FUNCTION_BLOCK FB_SLIDERLR (* FB_SLIDER with local publication of REAL position *)
  (* Standard: 61499-1; Classification: HMI *)
  (* Version 0.0, 2006-11-15, JHC, Holobloc Inc, Copied/Modified from FB_SLIDERL. *)
  (* Compiler header: package fb.rt.hmi; import fb.rt.mva.FBMVCD; import fb.rt.net.*; import fb.rt.math.*; *)
  (* Compiler classdef: public class FB_SLIDERLR extends FBMVCD *)
  (* Compiler Java Sun JDK 1.5.0 *)
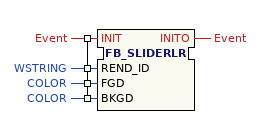
  EVENT_INPUT
    INIT WITH REND_ID, BKGD, FGD; (* Initialization Request *)
  END_EVENT
  EVENT_OUTPUT
    INITO; (* Initialization Confirm *)
  END_EVENT
  VAR_INPUT
    REND_ID : WSTRING; (* Data Channel ID - default is FB instaqnce name *)
    FGD : COLOR := red; (* Slider Foreground Color *)
    BKGD : COLOR := blue; (* Slider Background Color *)
  END_VAR
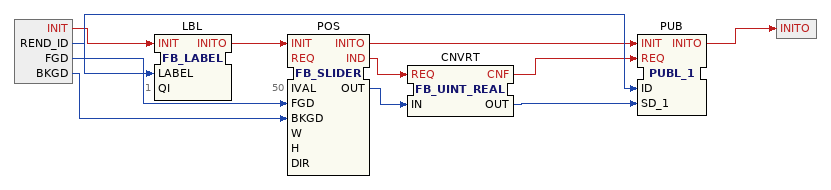
  FBS
    LBL : FB_LABEL(QI := 1);
    POS : FB_SLIDER(IVAL := 50);
    PUB : PUBL_1;
    CNVRT : FB_UINT_REAL;
  END_FBS
  EVENT_CONNECTIONS
    INIT TO LBL.INIT;
    LBL.INITO TO POS.INIT;
    PUB.INITO TO INITO;
    POS.INITO TO PUB.INIT;
    POS.IND TO CNVRT.REQ;
    CNVRT.CNF TO PUB.REQ;
  END_CONNECTIONS
  DATA_CONNECTIONS
    REND_ID TO PUB.ID;
    REND_ID TO LBL.LABEL;
    FGD TO POS.FGD;
    BKGD TO POS.BKGD;
    POS.OUT TO CNVRT.IN;
    CNVRT.OUT TO PUB.SD_1;
  END_CONNECTIONS
END_FUNCTION_BLOCK
